// TIA Portal V17 export
// export: Created 2025-04-11T04:54:24.1963426Z, ExportSetting WithDefaults, DisplayName Totally Integrated Automation Portal, DisplayVersion V17, DisplayName TIA Portal Openness, DisplayVersion V17, DisplayName TIA Portal Version Control Interface, DisplayVersion V17, DisplayName SINAMICS Startdrive Advanced, DisplayVersion V17, DisplayName SINAMICS Startdrive G130, G150, S120, S150, SINAMICS MV, S210, DisplayVersion V17, DisplayName SINAMICS Startdrive G110M, G120, G120C, G120D, G120P, G115D, DisplayVersion V17, DisplayName STEP 7 Professional, DisplayVersion V17, DisplayName STEP 7 Safety, DisplayVersion V17, DisplayName WinCC Advanced, DisplayVersion V17
TYPE "UDT_Device_Keep"
// stored: IsFailsafeCompliant false
   STRUCT
      IN_tStartTime : Time := T#10S;   // 启动设备超时时间
      IN_tStopTime : Time := T#10S;   // 停止设备超时时间
      IN_xAlarmEnable : Bool := TRUE;   // 报警使能
      OUT_tCurrentRun : UDInt;   // 本次运行时间(分钟)
   END_STRUCT;
END_TYPE
